(* CODESYS project CannyIEC
   Author: Roy Ratcliffe
   Company: Roy Ratcliffe
   DefaultNamespace: CANNY
   Description: Library project template with all possible element types, docu and a sample project structure
   DocFormat: reStructuredText
   LanguageModelAttribute: qualified-access-only
   Placeholder: CannyIEC
   Title: CannyIEC Library
   Version: 0.1.5.2

Project tree, tasks and I/O mapping:
  CannyIEC/
    GlobalVariables/
      global variables Variables
  function GetLibVersion [ST]
  function GetLibVersionNumber [ST]
  function IsLibReleased [ST]
  data type ERROR
  function block AsymmetricDebounce [ST]
  function block FirstCycle [ST]
  function block PT1 [ST]
  function block SymmetricDebounce [ST]
  function block TRIG [ST]
  function ISIGNBIT [ST]
  function REPSILONEQ [ST]
  function RSIGNBIT [ST]
  global variables Constants
*)

// ERROR
{attribute 'qualified_only'}
//{attribute 'conditionalshow'}
//{attribute 'conditionalshow' := 'SomeText'}
//{attribute 'hide'}
TYPE ERROR : (
        NO_ERROR,
        TIME_OUT
    );
END_TYPE

// Constants
{attribute 'qualified_only'}
//{attribute 'conditionalshow'}
//{attribute 'conditionalshow' := 'SomeText'}
//{attribute 'hide'}
VAR_GLOBAL CONSTANT
    gc_iDummy : INT := 42; /// This is a dummy global constant variable
END_VAR

// CannyIEC/GlobalVariables/Variables
{attribute 'qualified_only'}
//{attribute 'conditionalshow'}
//{attribute 'conditionalshow' := 'SomeText'}
//{attribute 'hide'}
VAR_GLOBAL
    g_iDummy : INT; /// This is a dummy global variable
END_VAR

// GetLibVersion
// This function has been automatically generated from the project information.
FUNCTION GetLibVersion : VERSION
VAR_INPUT
	
END_VAR

GetLibVersion.uiMajor := 0;
GetLibVersion.uiMinor := 1;
GetLibVersion.uiServicePack := 11;
GetLibVersion.uiPatch := 10;

END_FUNCTION

// GetLibVersionNumber
// This function has been automatically generated from the project information.
FUNCTION GetLibVersionNumber : DWORD
VAR_INPUT
	
END_VAR

GetLibVersionNumber := 68362;

END_FUNCTION

// IsLibReleased
// This function has been automatically generated from the project information.
FUNCTION IsLibReleased : BOOL
VAR_INPUT
	
END_VAR

IsLibReleased := FALSE;

END_FUNCTION

// AsymmetricDebounce
FUNCTION_BLOCK AsymmetricDebounce
VAR_INPUT
    IN          : BOOL;           (* raw input signal from a sensor or switch *)
    tPresetRise : TIME := T#50MS; (* preset time for rising edge debounce *)
    tPresetFall : TIME := T#50MS; (* preset time for falling edge debounce *)
END_VAR
VAR_OUTPUT
    Q : BOOL; (* debounced "input" signal *)
END_VAR
VAR
    fbDebounce : TON;
END_VAR

(* Only accept a state change after the raw input remains stable for its
   configured debounce time. The input must remain stable for the
   specified debounce time before the output changes. The TON's input
   receives the XOR of the raw input and the current output, ensuring
   that the timer only runs when there is a state change. *)
fbDebounce(IN := IN <> Q, PT := SEL(IN, tPresetFall, tPresetRise));
IF fbDebounce.Q THEN
    Q := IN;
END_IF;

END_FUNCTION_BLOCK

// FirstCycle
FUNCTION_BLOCK FirstCycle
VAR_OUTPUT
    Q : BOOL; (* TRUE during the first cycle of the program run *)
END_VAR
VAR
    X : BOOL := FALSE; (* Has executed at least once during the program run *)
END_VAR

(* Track the first cycle of the program run. Q will be TRUE only during
   the first cycle, and X will be set to TRUE afterwards. *)
Q := NOT X;
X := TRUE;

END_FUNCTION_BLOCK

// PT1
FUNCTION_BLOCK PT1
VAR_INPUT
    IN : REAL; (* Input signal *)
END_VAR
VAR_OUTPUT
    Q1 : REAL; (* Output signal *)
END_VAR
VAR_INPUT
    P : REAL; (* Proportional factor *)
END_VAR
VAR
    P1 : REAL; (* Limited proportional factor *)
    Q  : REAL; (* Previous output signal, used for feedback *)
END_VAR

(* First, limit the proportional factor to the range [0, 1] because
values outside this range could lead to instability or unexpected
behaviour. Next, calculate the output signal using the limited
proportional factor and the internal state, i.e. the previous output
signal. The current cycle's output becomes the next cycle's feedback.

Avoid SA0038: read access to output variable within the same cycle. IEC
61131-3 standard recommends avoiding read access to output variables
within the same cycle. It is considered a bad practice and can lead to
unpredictable behavior in the control logic. *)
P1 := LIMIT(0, P, 1);
Q  := (IN * P1) + (Q * (1 - P1));
Q1 := Q;

END_FUNCTION_BLOCK

// SymmetricDebounce
FUNCTION_BLOCK SymmetricDebounce
VAR_INPUT
    xDirty : BOOL; (* raw input signal from a sensor or switch *)
END_VAR
VAR_OUTPUT
    xClean : BOOL; (* debounced "input" signal *)
END_VAR
VAR
    tPresetRising    : TIME;           (* preset time for rising edge debounce *)
    tPresetFalling   : TIME;           (* preset time for falling edge debounce *)
    tPreset          : TIME := T#50MS; (* symmetric preset time used if specific rising/falling presets are not set; default to 50 milliseconds *)
    fbDelayedRising  : TON;            (* timer for rising edge *)
    fbDelayedFalling : TOF;            (* timer for falling edge *)
END_VAR

(* The raw input signal passes through the TON and TOF function blocks, which
implement the debounce logic. The TON block starts timing when the raw input
goes high, and the TOF block starts timing when the TON output goes low. The
system takes the debounced output signal from the TOF output. *)
(* Rising edge debounce *)
fbDelayedRising(IN := xDirty, PT := SEL(tPresetRising <> T#0S, tPresetRising, tPreset));
(* Falling edge debounce *)
fbDelayedFalling(IN := fbDelayedRising.Q, PT := SEL(tPresetFalling <> T#0S, tPresetFalling, tPreset));
xClean := fbDelayedFalling.Q;

END_FUNCTION_BLOCK

// TRIG
FUNCTION_BLOCK TRIG
VAR_INPUT
    CLK : BOOL; (* signal to monitor *)
END_VAR
VAR_OUTPUT
    Q : BOOL; (* one-cycle pulse when CLK changes *)
END_VAR
VAR
    fbRise : R_TRIG; (* rising edge trigger *)
    fbFall : F_TRIG; (* falling edge trigger *)
END_VAR

fbRise(CLK := CLK);
fbFall(CLK := CLK);
Q := fbRise.Q OR fbFall.Q;

END_FUNCTION_BLOCK

// ISIGNBIT
FUNCTION ISIGNBIT : BIT
VAR_INPUT
    iValue : INT;
END_VAR

ISIGNBIT := iValue < INT#0;

END_FUNCTION

// REPSILONEQ
FUNCTION REPSILONEQ : BOOL
VAR_INPUT
    rLHS     : REAL;              (* nominal left-hand side *)
    rRHS     : REAL;              (* nominal right-hand side *)
    rEpsilon : REAL := REAL#1e-6; (* allowable difference *)
END_VAR

(* Error band is inclusive of the epsilon value.
Less than or equal to is close enough, rather than strict equality. *)
REPSILONEQ := ABS(rLHS - rRHS) <= rEpsilon;

END_FUNCTION

// RSIGNBIT
FUNCTION RSIGNBIT : BIT
VAR_INPUT
    rValue : REAL;
END_VAR

RSIGNBIT := rValue < REAL#0;

END_FUNCTION
